// TIA Portal V20 export
FUNCTION_BLOCK "定位轴基本控制"   // FB1, LAD
{ S7_Optimized_Access := 'TRUE' }
// stored: MemoryReserve 100, SetENOAutomatically false
   VAR_INPUT
      轴号 : TO_PositioningAxis;
      使能 : Bool;
      回原 : Bool;
      回原模式 : Int;
      绝对定位 : Bool;
      相对定位 : Bool;
      暂停 : Bool;
      复位 : Bool;
      绝对位置 : Real;
      绝对速度 : Real;
      相对位置 : Real;
      相对速度 : Real;
      点动正转 : Bool;
      点动反转 : Bool;
      点动速度 : Real;
   END_VAR
   VAR_OUTPUT
      轴已启用 : Bool;
      使能错误 : Bool;
      回原完成 : Bool;
      回原错误 : Bool;
      绝对定位完成 : Bool;
      绝对定位错误 : Bool;
      相对定位完成 : Bool;
      相对定位错误 : Bool;
      点动中 : Bool;
      点动错误 : Bool;
      当前位置 : Real;
      当前速度 : Real;
   END_VAR
   VAR
      MC_Power_Instance { S7_SetPoint := 'True'} : MC_Power;
      MC_Home_Instance { S7_SetPoint := 'True'} : MC_Home;
      MC_MoveAbsolute_Instance { S7_SetPoint := 'True'} : MC_MoveAbsolute;
      MC_MoveRelative_Instance { S7_SetPoint := 'True'} : MC_MoveRelative;
      MC_Reset_Instance { S7_SetPoint := 'True'} : MC_Reset;
      MC_Halt_Instance { S7_SetPoint := 'True'} : MC_Halt;
      MC_MoveJog_Instance { S7_SetPoint := 'True'} : MC_MoveJog;
   END_VAR
   VAR_TEMP
      复位完成 : Bool;
      复位错误 : Bool;
      暂停完成 : Bool;
      暂停错误 : Bool;
   END_VAR
   VAR_TEMP   // added for the SCL form of the ladder/FBD networks
      _w1 : Bool;
      _w2 : Bool;
      _w3 : Bool;
   END_VAR
BEGIN

REGION Network 1
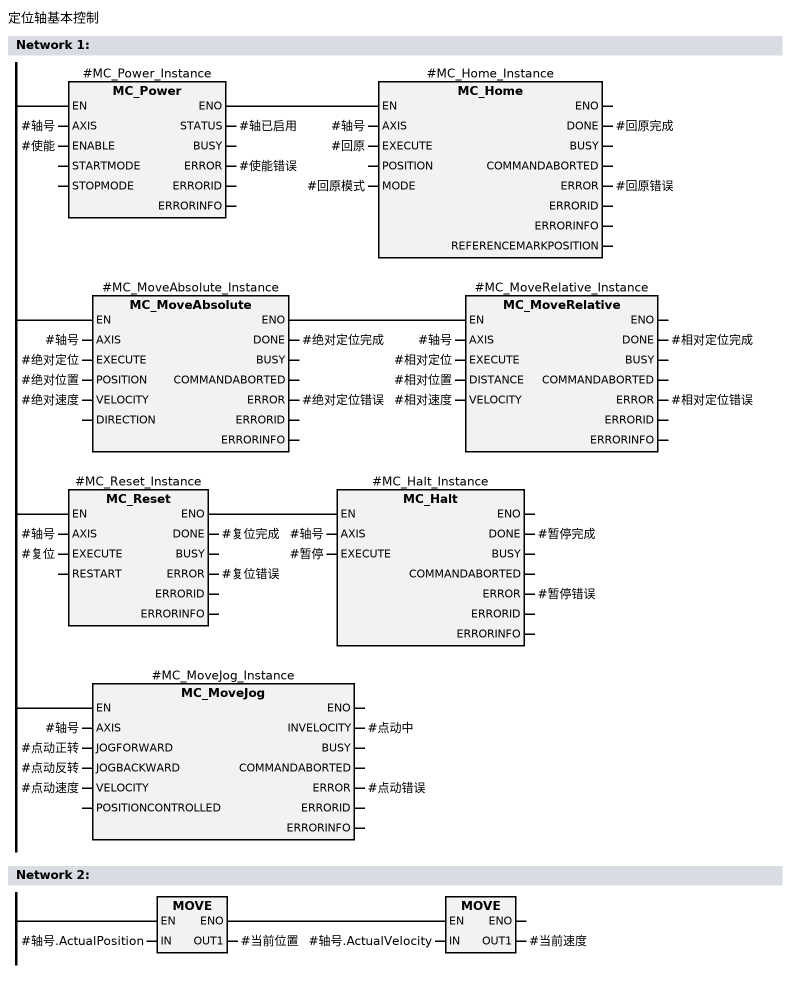
   RUNG wire#powerrail
      #MC_Power_Instance.MC_Power(Axis := #轴号, Enable := #使能, StartMode :=, StopMode :=, Status => #轴已启用, Busy =>, Error => #使能错误, ErrorID =>, ErrorInfo =>)
      #MC_Home_Instance.MC_Home(Axis := #轴号, Execute := #回原, Position :=, Mode := #回原模式, Done => #回原完成, Busy =>, CommandAborted =>, Error => #回原错误, ErrorID =>, ErrorInfo =>, ReferenceMarkPosition =>)
   END_RUNG
   RUNG wire#powerrail
      #MC_MoveAbsolute_Instance.MC_MoveAbsolute(Axis := #轴号, Execute := #绝对定位, Position := #绝对位置, Velocity := #绝对速度, Direction :=, Done => #绝对定位完成, Busy =>, CommandAborted =>, Error => #绝对定位错误, ErrorID =>, ErrorInfo =>)
      #MC_MoveRelative_Instance.MC_MoveRelative(Axis := #轴号, Execute := #相对定位, Distance := #相对位置, Velocity := #相对速度, Done => #相对定位完成, Busy =>, CommandAborted =>, Error => #相对定位错误, ErrorID =>, ErrorInfo =>)
   END_RUNG
   RUNG wire#powerrail
      #MC_Reset_Instance.MC_Reset(Axis := #轴号, Execute := #复位, Restart :=, Done => #复位完成, Busy =>, Error => #复位错误, ErrorID =>, ErrorInfo =>)
      #MC_Halt_Instance.MC_Halt(Axis := #轴号, Execute := #暂停, Done => #暂停完成, Busy =>, CommandAborted =>, Error => #暂停错误, ErrorID =>, ErrorInfo =>)
   END_RUNG
   RUNG wire#powerrail
      #MC_MoveJog_Instance.MC_MoveJog(Axis := #轴号, JogForward := #点动正转, JogBackward := #点动反转, Velocity := #点动速度, PositionControlled :=, InVelocity => #点动中, Busy =>, CommandAborted =>, Error => #点动错误, ErrorID =>, ErrorInfo =>)
   END_RUNG
   // the same network as SCL:
   #MC_Power_Instance(Axis := #轴号, Enable := #使能, Status => #轴已启用, Error => #使能错误, ENO => #_w1);   // MC_Power
   IF #_w1 THEN
       #MC_Home_Instance(Axis := #轴号, Execute := #回原, Mode := #回原模式, Done => #回原完成, Error => #回原错误);   // MC_Home
   END_IF;
   #MC_MoveAbsolute_Instance(Axis := #轴号,   // MC_MoveAbsolute
                           Execute := #绝对定位,
                           Position := #绝对位置,
                           Velocity := #绝对速度,
                           Done => #绝对定位完成,
                           Error => #绝对定位错误,
                           ENO => #_w2);
   IF #_w2 THEN
       #MC_MoveRelative_Instance(Axis := #轴号,   // MC_MoveRelative
                               Execute := #相对定位,
                               Distance := #相对位置,
                               Velocity := #相对速度,
                               Done => #相对定位完成,
                               Error => #相对定位错误);
   END_IF;
   #MC_Reset_Instance(Axis := #轴号, Execute := #复位, Done => #复位完成, Error => #复位错误, ENO => #_w3);   // MC_Reset
   IF #_w3 THEN
       #MC_Halt_Instance(Axis := #轴号, Execute := #暂停, Done => #暂停完成, Error => #暂停错误);   // MC_Halt
   END_IF;
   #MC_MoveJog_Instance(Axis := #轴号,   // MC_MoveJog
                        JogForward := #点动正转,
                        JogBackward := #点动反转,
                        Velocity := #点动速度,
                        InVelocity => #点动中,
                        Error => #点动错误);
END_REGION

REGION Network 2
   RUNG wire#powerrail
      Move(in := #轴号.ActualPosition, out1 => #当前位置)
      Move(in := #轴号.ActualVelocity, out1 => #当前速度)
   END_RUNG
   // the same network as SCL:
   #当前位置 := #轴号.ActualPosition;
   #当前速度 := #轴号.ActualVelocity;
END_REGION
END_FUNCTION_BLOCK
